Staubli VAL3: cycle_resume.pgx

program cycle_resume()
begin
  // resume from PAUSE
  if cycleStatus:bPause==true
    //raise the bit
    cycleStatus:bToPause=true
    watch(cycleStatus:bToPause==false,1)
    // OnEvent
    call OnEvent:OnCycleEvent(3)
  endIf
end
